TYPE TAC_Standard :
STRUCT
	MesData : TAC; 			(* Main Structure *)
END_STRUCT
END_TYPE

(* stored: Version 1.1.0.1, ProductVersion 3.1.4024.11
   DUT TAC_Standard: Id {3422510f-35ba-4005-b48a-b55fbc605f45} *)
